// TwinCAT 3 PLC project PLCSim
// ProgramVersion: 3.1.4022.3
// libraries:
//   Tc2_Standard, * (Beckhoff Automation GmbH)
//   Tc2_System, * (Beckhoff Automation GmbH)
//   Tc3_Module, * (Beckhoff Automation GmbH)
// project tree:
//   / GlobalTextList.TcGTLO, PlcTask.TcTTO, Visualization Manager.TcVMO (not stored)
//   GVLs/ GVL.TcGVL
//   POUs/ MAIN.TcPOU
//   VISUs/ Visualization.TcVIS

CONFIGURATION PLCSim
    RESOURCE PLC ON TwinCAT3
        TASK PlcTask(INTERVAL := T#80ms, PRIORITY := 1);
        PROGRAM MAIN WITH PlcTask : MAIN;
    END_RESOURCE
END_CONFIGURATION

// ---- GVLs/GVL.TcGVL
{attribute 'qualified_only'}
VAR_GLOBAL
	qxPulseOne		AT %Q*:	BOOL; 		(* PULS button *)
	qxStart			AT %Q*:	BOOL; 		(* START switch *)
	qxSetLevel		AT %Q*:	BOOL; 		(* NIVÅ switch *)
	qxLevel3		AT %Q*:	BOOL; 		(* Sensor for level 3 *)
	qxLevel2		AT %Q*:	BOOL; 		(* Sensor for level 2 *)
	qxLevel1		AT %Q*:	BOOL; 		(* Sensor for level 1 *)
	qxNotEmpty		AT %Q*:	BOOL; 		(* Sensor for not empty *)
	qxTempOk		AT %Q*:	BOOL; 		(* Temp sensor *)
	qwCurTemp		AT %Q*: INT:=20;	(* Current Temparature *)
	qwSetTem		AT %Q*:	INT:= 40;	(* Setting temparature Button *)
	
	ixPulseTwo		AT %I*:	BOOL; 		(* PULS button *)
	ixForw			AT %I*:	BOOL; 		(* Washer cylinder forward *)
	ixBack			AT %I*:	BOOL; 		(* Washer cylinder back *)
	ixSpin			AT %I*:	BOOL; 		(* Washer cylinder spin *)
	ixHeating		AT %I*:BOOL;		(* Heating coil ON *)
	ixFill			AT %I*:	BOOL; 		(* Fill water *)
	ixDrain			AT %I*:	BOOL; 		(* Drain water *)
	ixDispBit1		AT %I*:	BOOL; 		(* Display bit 1 *)
	ixDispBit2		AT %I*:	BOOL; 		(* Display bit 2 *)

	nWaterLev:		INT:=0;			(* Internal variable *)
	nShowWater:		INT;			(* Internal variable *)
	nDispNo:		INT:=0;			(* Internal variable *)
	nCylPos:		INT:=0;			(* Internal variable *)

END_VAR

// ---- POUs/MAIN.TcPOU
PROGRAM MAIN
VAR
END_VAR

VAR CONSTANT
	WaterLevMax:		INT:= 200;
	WaterLev3:			INT:= 150;
	WaterLev2:			INT:= 100;
	WaterLev1:			INT:= 50;
END_VAR

(*  function block Washer  *)
(*  2008-10-08  BoS University West *)
(*	2023-02-17	GabrielS	Updated to GVL and Exam Version*)

(*  -------------  water level  -----------------  *)
IF GVL.ixFill AND GVL.nWaterLev < WaterLevMax THEN				(* increase water level *)
	GVL.nWaterLev := GVL.nWaterLev + 1;
END_IF

IF GVL.ixDrain AND GVL.nWaterLev > 0 THEN						(* decrease water level *)
	GVL.nWaterLev := GVL.nWaterLev - 1;
END_IF

GVL.nShowWater := - GVL.nWaterLev;								(* inverting only for display function *)

(*  -------------  water level sensors  -----------------  *)
IF GVL.nWaterLev > 0 THEN
	GVL.qxNotEmpty := TRUE;
ELSE
	GVL.qxNotEmpty := FALSE;
END_IF
IF GVL.nWaterLev >= WaterLev1 THEN
	GVL.qxLevel1 := TRUE;
ELSE
	GVL.qxLevel1 := FALSE;
END_IF
IF GVL.nWaterLev >= WaterLev2 THEN
	GVL.qxLevel2 := TRUE;
ELSE
	GVL.qxLevel2 := FALSE;
END_IF
IF GVL.nWaterLev >= WaterLev3 THEN
	GVL.qxLevel3 := TRUE;
ELSE
	GVL.qxLevel3 := FALSE;
END_IF


(*  -------------  water temp sensor  -----------------  *)

IF GVL.qwCurTemp > GVL.qwSetTem-3 AND GVL.qwCurTemp < GVL.qwSetTem+3 THEN
	GVL.qxTempOk := TRUE;
ELSE
	GVL.qxTempOk := FALSE;
END_IF

(*  -----------  Water Heater and Cooler  -------------  *)

IF gvl.ixHeating AND GVL.qwCurTemp < 100 THEN
	gvl.qwCurTemp:=gvl.qwCurTemp+1;
ELSIF NOT gvl.ixHeating AND GVL.qwCurTemp > 2 THEN
	gvl.qwCurTemp:=gvl.qwCurTemp-1;
END_IF

(*  -------------  cylinder posistion  -----------------  *)
IF GVL.ixForw AND NOT GVL.ixSpin THEN
	GVL.nCylPos := GVL.nCylPos+5;
ELSIF GVL.ixForw AND GVL.ixSpin THEN
	GVL.nCylPos := GVL.nCylPos+15;
END_IF
IF GVL.ixBack AND NOT GVL.ixSpin THEN
	GVL.nCylPos := GVL.nCylPos-5;
ELSIF GVL.ixBack AND  GVL.ixSpin THEN
	GVL.nCylPos := GVL.nCylPos-15;
END_IF

IF GVL.nCylPos > 359 THEN
	GVL.nCylPos := 0;
ELSIF GVL.nCylPos < 0 THEN
	GVL.nCylPos :=355;
END_IF

(*  -------------  display number  -----------------  *)
IF NOT GVL.ixDispBit1 AND NOT GVL.ixDispBit2 THEN
	GVL.nDispNo:=0;
ELSIF GVL.ixDispBit1 AND NOT GVL.ixDispBit2 THEN
	GVL.nDispNo:=1;
ELSIF NOT GVL.ixDispBit1 AND  GVL.ixDispBit2 THEN
	GVL.nDispNo:=2;
ELSIF GVL.ixDispBit1 AND GVL.ixDispBit2 THEN
	GVL.nDispNo:=3;
END_IF

END_PROGRAM

// ---- GlobalTextList.TcGTLO
TEXTLIST GlobalTextList
  464 = '  LEVEL\n     HIGH                   NORM'
  992 = '  LEVEL\n     HIGH                 NORM'
  506 = '  LEVEL\n   HIGH                   NORM'
  798 = '  LEVEL\n   HIGH                 NORM'
  928 = '  LEVEL\nHIGH                   NORM'
  916 = '  LEVEL\nHIGHT                   NORM'
  815 = '  LEVEL\nNORM                   HIGH'
  391 = '  START                 STOP'
  709 = '  START               STOP'
  882 = '  START             STOP'
  762 = '  START            STOP'
  113 = '  START           STOP'
  77 = '  STOP                  START'
  5 = '%i'
  526 = 'CUR TEMP'
  6 = 'DISPLAY'
  821 = 'LEVEL\nNORM                   HIGH'
  463 = 'Level 1'
  805 = 'Level 2'
  694 = 'Level 3'
  236 = 'Level Not Emty'
  825 = 'NORM '
  830 = 'Puls'
  172 = 'PULS'
  549 = 'PULS ONE'
  377 = 'PULS TWO'
  7 = 'SET TEMP'
  556 = 'Temp OK'
  910 = 'TEMP OK'
  141 = 'University West\nAnders N Dec 2018'
  460 = 'University West\nATM700 Exam Feb2023'
  965 = 'University West \nAnders Nilsson\nATM700 Exam Feb2023'
END_TEXTLIST

// ---- VISUs/Visualization.TcVIS
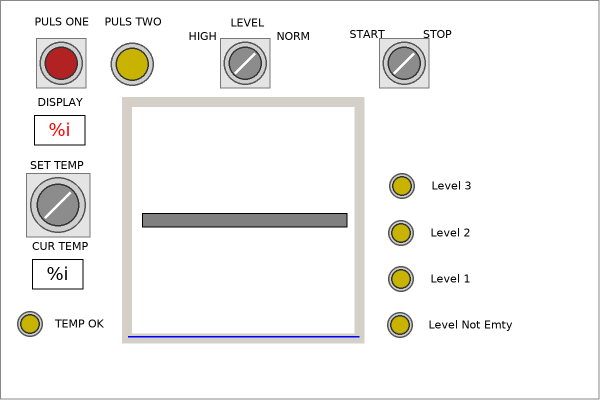
VISUALIZATION Visualization  // 600x400
    Rectangle (122,97 242x246)
    PushSwitch (36,38 50x50), variable: GVL.qxPulseOne, behaviour: TOGGLE, style: Switch-PushSwitch-Red
    Label (10,11 104x22), "PULS ONE"
    RotarySwitch (220,38 50x50), variable: GVL.qxSetLevel, input disabled if: GVL.qxStart, behaviour: TOGGLE, style: Switch-RotarySwitch-Gray
    Label (164,10 160x39), "LEVEL HIGH NORM"
    RotarySwitch (379,38 50x50), variable: GVL.qxStart, behaviour: TOGGLE, style: Switch-RotarySwitch-Gray
    Label (317,15 160x39), "START STOP"
    Lamp1 (387,171 30x30), variable: GVL.qxLevel3, style: Lamp-Lamp1-Yellow
    Label (420,178 63x16), "Level 3"
    Lamp1 (386,218 30x30), variable: GVL.qxLevel2, style: Lamp-Lamp1-Yellow
    Label (419,225 63x16), "Level 2"
    Lamp1 (386,264 30x30), variable: GVL.qxLevel1, style: Lamp-Lamp1-Yellow
    Label (419,271 63x16), "Level 1"
    Lamp1 (385,310 30x30), variable: GVL.qxNotEmpty, style: Lamp-Lamp1-Yellow
    Label (418,317 105x16), "Level Not Emty"
    Lamp1 (15,309 30x30), variable: GVL.qxTempOk, style: Lamp-Lamp1-Yellow
    Label (48,316 63x16), "TEMP OK"
    Potentiometer360 (24,173 68x64), variable: GVL.qwSetTem, style: Potentiometer-Potentiometer360-Gray, scale format: %i, scale 0..100
        p2431819421: Outside
    Rectangle (32,259 51x30), "%i", text variable: GVL.qwCurTemp
    Label (14,237 92x19), "CUR TEMP"
    Label (11,156 92x19), "SET TEMP"
    Label (14,93 92x19), "DISPLAY"
    Rectangle (34,115 51x30), "%i", text variable: GVL.qwSetTem
    Rectangle (128,336 231x1)
        p2773130477: GVL.nShowWater
    Rectangle (142,213 205x14)
        p2858320360: GVL.nCylPos
    Label (81,11 104x22), "PULS TWO"
    Lamp1 (107,39 50x50), variable: GVL.ixPulseTwo, style: Lamp-Lamp1-Yellow
END_VISUALIZATION
